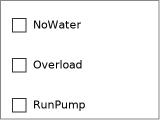
VISUALIZATION Vi_Sim_TankCtrl  // 160x120
VAR_IN_OUT
	obj			: TankCtrl;
END_VAR
    Checkbox (10,10 150x30), "NoWater", variable: obj.bNoWater
    Checkbox (10,50 150x30), "Overload", variable: obj.bOverload
    Checkbox (10,90 150x30), "RunPump", variable: obj.bRunPump
END_VISUALIZATION

(* stored: Version 1.1.0.1
   Visu Vi_Sim_TankCtrl: Id {b3761375-64da-4cad-9dfb-4a7e01ccc40c} *)
